% RSLogix 500 project HEATER_ANALOG_BAK003.RSS, saved by version 8.30.00.16 %
PROJECT "UNTITLED"    % processor: Bul.1763 MicroLogix 1100 Series B %

PROGRAM FILES
  LAD 2 "MAIN"  6 rungs

DATA FILES
  O0 OUTPUT  8 elements
  I1 INPUT  16 elements
  S2 STATUS  66 elements
  B3 BINARY  1 elements
  T4 TIMER  1 elements
  C5 COUNTER  1 elements
  R6 CONTROL  1 elements
  N7 INTEGER  2 elements
  F8 FLOAT  1 elements
  PD9 TEMP  1 elements

LADDER 2 "MAIN"
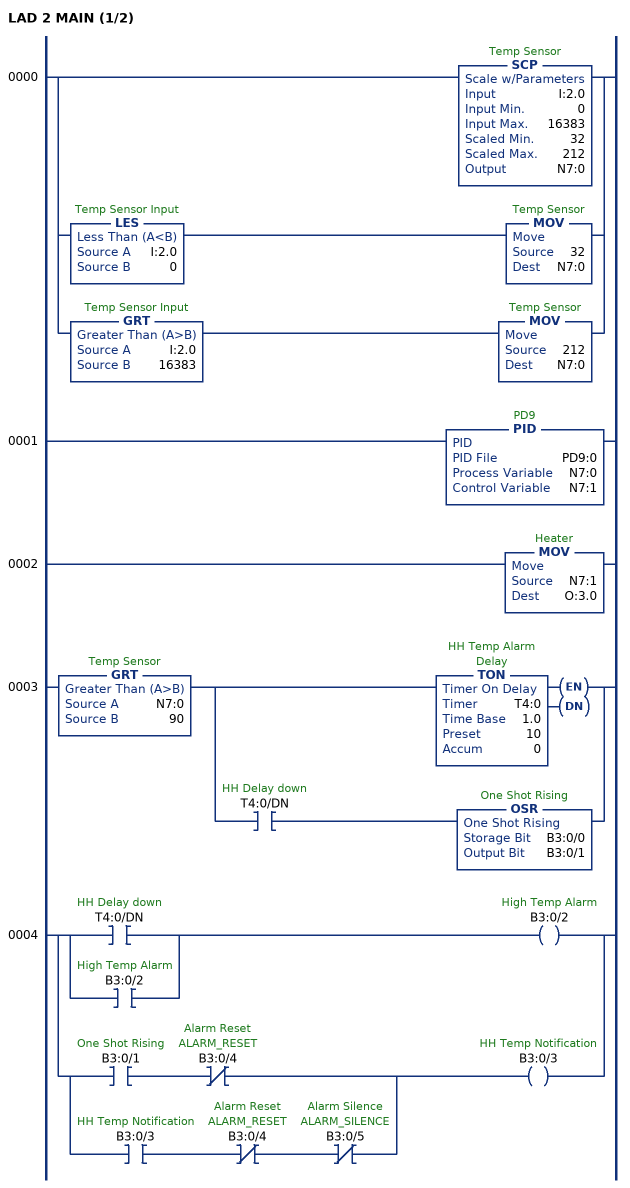
% Rung: 0 %
SOR BST SCP I:2.0 0 16383 32 212 N7:0 NXB LES I:2.0 0 MOV 32 N7:0 NXB GRT I:2.0 16383 MOV 212 N7:0 BND EOR
%   I:2.0  "Temp Sensor Input" %
%   N7:0  "Temp Sensor" %
% Rung: 1 %
SOR PID PD9:0 N7:0 N7:1 EOR
%   PD9:0  PD9 %
%   N7:0  "Temp Sensor" %
%   N7:1  "PID Output" %
% Rung: 2 %
SOR MOV N7:1 O:3.0 EOR
%   N7:1  "PID Output" %
%   O:3.0  "Heater" %
% Rung: 3 %
SOR GRT N7:0 90 BST TON T4:0 1.0 10 0 NXB XIC T4:0/DN OSR B3:0/0 B3:0/1 BND EOR
%   N7:0  "Temp Sensor" %
%   T4:0  "HH Temp Alarm Delay" %
%   T4:0/DN  "HH Delay down" %
%   B3:0/0  "One Shot Rising" %
%   B3:0/1  "One Shot Rising" %
% Rung: 4 %
SOR BST BST XIC T4:0/DN NXB XIC B3:0/2 BND OTE B3:0/2 NXB BST XIC B3:0/1 XIO B3:0/4 NXB XIC B3:0/3 XIO B3:0/4 XIO B3:0/5 BND OTE B3:0/3 BND EOR
%   T4:0/DN  "HH Delay down" %
%   B3:0/2  "High Temp Alarm" %
%   B3:0/1  "One Shot Rising" %
%   B3:0/4  ALARM_RESET  "Alarm Reset" %
%   B3:0/3  "HH Temp Notification" %
%   B3:0/5  ALARM_SILENCE  "Alarm Silence" %

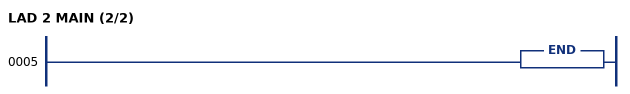
% Rung: 5 %
SOR END EOR

OTHER DOCUMENTED ADDRESSES
  N7:1/0  "Temp Controller"
  O:3.0/0  "Output"

DATA TABLE (non-zero values as saved)
DATA T4
% .PRE .ACC %
% T4:0 % 10 0
